KUKA KRL program: toolsetup.src, toolsetup.dat

--- toolsetup.src ---
&ACCESS RVO
&REL 3
&PARAM EDITMASK = *
&PARAM TEMPLATE = C:\KRC\Roboter\Template\vorgabe
DEF toolsetup( )

   BAS (#INITMOV,0)
ptp $pos_act

   MoveSettings(9, 10, 100, 100)
lin {x 160 ,y 160,z 10, a 0, b 0,c 0}
END

--- toolsetup.dat ---
&ACCESS RVO
&REL 3
&PARAM EDITMASK = *
&PARAM TEMPLATE = C:\KRC\Roboter\Template\vorgabe
DEFDAT toolsetup
;FOLD EXTERNAL DECLARATIONS;%{PE}%MKUKATPBASIS,%CEXT,%VCOMMON,%P
;FOLD BASISTECH EXT;%{PE}%MKUKATPBASIS,%CEXT,%VEXT,%P
EXT  BAS (BAS_COMMAND  :IN,REAL  :IN )
DECL INT SUCCESS
;ENDFOLD (BASISTECH EXT)
;FOLD USER EXT;%{E}%MKUKATPUSER,%CEXT,%VEXT,%P
;Make your modifications here

;ENDFOLD (USER EXT)
;ENDFOLD (EXTERNAL DECLARATIONS)
ENDDAT
